// TIA Portal project "Anderca_Mihai_Teodor_Aplicatie_Practica_AIA_Licenta" (V15.1)

(* hardware
DEVICE "S7-1200 station_1"  S7-1200 Station
   slot 0: "Rack_0"  S7-1200 Rack  Rack  V1.0
   slot 1: "PLC_1"  CPU 1215C AC/DC/Rly  6ES7 215-1BG40-0XB0  V4.2
*)

// ===== PLC "PLC_1"  CPU 1215C AC/DC/Rly =====

VAR_GLOBAL   // PLC tag table "Palletizer tag table"
   "Transporto Role Incarcare Palet" AT %Q1.5 : Bool;
   "Tag_1" AT %M0.0 : Bool;
   "Senzor Palet Spate" AT %I5.2 : Bool;
   "Senzor Palet Fata" AT %I5.3 : Bool;
   "Lant Ascensor" AT %Q1.6 : Bool;
   "Senzor Palet Ridicat" AT %I5.6 : Bool;
   "Placa Deschisa" AT %M1.2 : Bool;
   "Palet Incarcat" AT %M1.4 : Bool;
   "Ascensor Ridicat" AT %Q1.7 : Bool;
   "Pusher" AT %Q2.1 : Bool;
   "Rand Complet Terminat" AT %M1.1 : Bool;
   "2 Cutii Incarcate" AT %M1.0 : Bool;
   "Banda Incarcare Cutii Incorporata" AT %Q2.3 : Bool;
   "Banda Incarcare Cutii" AT %Q2.5 : Bool;
   "Senzor Cutie Incarcata" AT %I5.4 : Bool;
   "Tag_6" AT %M0.3 : Bool;
   "Rand Incarcat" AT %M1.3 : Bool;
   "Tag_8" AT %M0.1 : Bool;
   "Cleste" AT %Q2.2 : Bool;
   "Deschidere Placa" AT %Q2.4 : Bool;
   "Placa Deschisa Maxim" AT %I5.5 : Bool;
   "Tag_9" AT %M0.4 : Bool;
   "Tag_10" AT %M1.6 : Bool;
   "Palet coborât" AT %M1.5 : Bool;
   "Coborare Palet" AT %Q2.0 : Bool;
   "Transportor Iesire" AT %Q2.6 : Bool;
   "Muta Ascensorul la Limita" AT %Q2.7 : Bool;
   "Tag_12" AT %M2.0 : Bool;
   "Tag_13" AT %M0.5 : Bool;
   "Tag_14" AT %M20.0 : Bool;
   "Placa Inchisa" AT %M3.0 : Bool;
   "Tag_16" AT %M3.1 : Bool;
   "Tag_17" AT %M3.2 : Bool;
   "Tag_18" AT %M0.6 : Bool;
   "Palet Gata de Coborâre" AT %M3.4 : Bool;
   "Palet Ridicat" AT %M3.6 : Bool;
END_VAR

VAR_GLOBAL   // PLC tag table "Sortare tag table"
   "Start Buton" AT %I4.0 : Bool;
   "Banda principala" AT %Q0.0 : Bool;
   "Banda Transportoare Stanga" AT %Q0.1 : Bool;
   "Banda Transportoare Dreapta" AT %Q0.2 : Bool;
   "Wheel Sorter" AT %Q0.4 : Bool;   // p
   "Deviere Stanga Wheel Sorter" AT %Q0.5 : Bool;
   "Deviere Dreapta Wheel Sorter" AT %Q0.6 : Bool;
   "Senzor cutie mica" AT %I4.1 : Bool;
   "Cutie Mica Detectata" AT %M30.0 : Bool;
   "Senzor Intrare Stanga" AT %I4.2 : Bool;
   "Cutie Mica Sortata" AT %M30.1 : Bool;
   "Senzor cutie mare" AT %I4.3 : Bool;
   "Senzor Intrare Dreapta" AT %I4.4 : Bool;
   "Cutie Mare Detectata" AT %M30.2 : Bool;
   "Cutie Mare Sortata" AT %M30.3 : Bool;
   "START" AT %M31.0 : Bool;
   "Start Led" AT %Q1.0 : Bool;
   "Stop Buton" AT %I4.5 : Bool;
   "STOP" AT %M31.1 : Bool;
   "Stop Led" AT %Q1.1 : Bool;
   "Banda Transportoare Inclinata" AT %Q0.7 : Bool;
END_VAR

VAR_GLOBAL CONSTANT   // PLC tag table "Sortare tag table"
   "None(1)" : Pip := 65535;
   "Automatic update(1)" : Pip := 0;
   "PIP 1(1)" : Pip := 1;
   "PIP 2(1)" : Pip := 2;
   "PIP 3(1)" : Pip := 3;
   "PIP 4(1)" : Pip := 4;
   "PIP OB Servo(1)" : Pip := 32768;
   "Local~MC(1)" : Hw_SubModule := 51;
   "Local~Common(1)" : Hw_SubModule := 50;
   "Local~Device(1)" : Hw_Device := 32;
   "Local~Configuration(1)" : Hw_SubModule := 33;
   "Local~Exec(1)" : Hw_SubModule := 52;
   "Local(1)" : Hw_SubModule := 49;
   "Local~PROFINET_interface_1(1)" : Hw_Interface := 64;
   "Local~PROFINET_interface_1~Port_1(1)" : Hw_Interface := 65;
   "Local~PROFINET_interface_1~Port_2(1)" : Hw_Interface := 66;
   "Local~HSC_1(1)" : Hw_Hsc := 257;
   "Local~HSC_2(1)" : Hw_Hsc := 258;
   "Local~HSC_3(1)" : Hw_Hsc := 259;
   "Local~HSC_4(1)" : Hw_Hsc := 260;
   "Local~HSC_5(1)" : Hw_Hsc := 261;
   "Local~HSC_6(1)" : Hw_Hsc := 262;
   "Local~AI_2_AQ_2_1(1)" : Hw_SubModule := 263;
   "Local~DI_14_DQ_10_1(1)" : Hw_SubModule := 264;
   "Local~Pulse_1(1)" : Hw_Pwm := 265;
   "Local~Pulse_2(1)" : Hw_Pwm := 266;
   "Local~Pulse_3(1)" : Hw_Pwm := 267;
   "Local~Pulse_4(1)" : Hw_Pwm := 268;
   "OB_Main(1)" : OB_PCYCLE := 1;
END_VAR

VAR_GLOBAL   // PLC tag table "PP tag table"
   "Senzor Amplasat" AT %I6.3 : Bool;
   "Senzor încorporat" AT %I6.4 : Bool;
   "Senzor Detecție Cutie deasupra Paletului" AT %I6.5 : Bool;
   "Transportor cu Role" AT %Q3.1 : Bool;
   "Prindere" AT %Q3.2 : Bool;
   "Deplasare Orizontală a Brațului" AT %Q3.3 : Bool;
   "Deplasare Verticală a Brațului" AT %Q3.4 : Bool;
   "Tag_7 pp" AT %M41.3 : Bool;
   "m41.4" AT %M41.5 : Bool;
   "Cutie detectată la Pick and Place" AT %M41.0 : Bool;
   "Tag_13 pp" AT %M41.1 : Bool;
   "Cutie Prinsă" AT %M41.2 : Bool;
   "Cutie deasupra Paletului" AT %M41.4 : Bool;
END_VAR

VAR_GLOBAL CONSTANT   // PLC tag table "PP tag table"
   "None(2)" : Pip := 65535;
   "Automatic update(2)" : Pip := 0;
   "PIP 1(2)" : Pip := 1;
   "PIP 2(2)" : Pip := 2;
   "PIP 3(2)" : Pip := 3;
   "PIP 4(2)" : Pip := 4;
   "PIP OB Servo(2)" : Pip := 32768;
   "Local~MC(2)" : Hw_SubModule := 51;
   "Local~Common(2)" : Hw_SubModule := 50;
   "Local~Device(2)" : Hw_Device := 32;
   "Local~Configuration(2)" : Hw_SubModule := 33;
   "Local~Exec(2)" : Hw_SubModule := 52;
   "Local(2)" : Hw_SubModule := 49;
   "Local~PROFINET_interface_1(2)" : Hw_Interface := 64;
   "Local~PROFINET_interface_1~Port_1(2)" : Hw_Interface := 65;
   "Local~PROFINET_interface_1~Port_2(2)" : Hw_Interface := 66;
   "Local~HSC_1(2)" : Hw_Hsc := 257;
   "Local~HSC_2(2)" : Hw_Hsc := 258;
   "Local~HSC_3(2)" : Hw_Hsc := 259;
   "Local~HSC_4(2)" : Hw_Hsc := 260;
   "Local~HSC_5(2)" : Hw_Hsc := 261;
   "Local~HSC_6(2)" : Hw_Hsc := 262;
   "Local~AI_2_AQ_2_1(2)" : Hw_SubModule := 263;
   "Local~DI_14_DQ_10_1(2)" : Hw_SubModule := 264;
   "Local~Pulse_1(2)" : Hw_Pwm := 265;
   "Local~Pulse_2(2)" : Hw_Pwm := 266;
   "Local~Pulse_3(2)" : Hw_Pwm := 267;
   "Local~Pulse_4(2)" : Hw_Pwm := 268;
   "OB_Main(2)" : OB_PCYCLE := 1;
END_VAR

// folder: System blocks/Program resources

DATA_BLOCK "IEC_Timer_0_DB"   // DB1
{ S7_Optimized_Access := 'TRUE' }
AUTHOR : Simatic
FAMILY : IEC
NAME : IEC_TMR
VERSION : 1.0
// stored: InstanceOfName IEC_TIMER
"IEC_TIMER"
BEGIN
END_DATA_BLOCK

DATA_BLOCK "IEC_Timer_0_DB_2"   // DB2
{ S7_Optimized_Access := 'TRUE' }
AUTHOR : Simatic
FAMILY : IEC
NAME : IEC_TMR
VERSION : 1.0
// stored: InstanceOfName IEC_TIMER
"IEC_TIMER"
BEGIN
END_DATA_BLOCK

DATA_BLOCK "IEC_Counter_0_DB"   // DB3
{ S7_Optimized_Access := 'TRUE' }
AUTHOR : Simatic
FAMILY : IEC
NAME : CNTR
VERSION : 1.0
// stored: InstanceOfName IEC_COUNTER
"IEC_COUNTER"
BEGIN
END_DATA_BLOCK

DATA_BLOCK "IEC_Timer_0_DB_1"   // DB4
{ S7_Optimized_Access := 'TRUE' }
AUTHOR : Simatic
FAMILY : IEC
NAME : IEC_TMR
VERSION : 1.0
// stored: InstanceOfName IEC_TIMER
"IEC_TIMER"
BEGIN
END_DATA_BLOCK

DATA_BLOCK "IEC_Counter_0_DB_1"   // DB5
{ S7_Optimized_Access := 'TRUE' }
AUTHOR : Simatic
FAMILY : IEC
NAME : CNTR
VERSION : 1.0
// stored: InstanceOfName IEC_COUNTER
"IEC_COUNTER"
BEGIN
END_DATA_BLOCK

DATA_BLOCK "IEC_Timer_0_DB_3"   // DB6
{ S7_Optimized_Access := 'TRUE' }
AUTHOR : Simatic
FAMILY : IEC
NAME : IEC_TMR
VERSION : 1.0
// stored: InstanceOfName IEC_TIMER
"IEC_TIMER"
BEGIN
END_DATA_BLOCK

DATA_BLOCK "IEC_Timer_0_DB_4"   // DB7
{ S7_Optimized_Access := 'TRUE' }
AUTHOR : Simatic
FAMILY : IEC
NAME : IEC_TMR
VERSION : 1.0
// stored: InstanceOfName IEC_TIMER
"IEC_TIMER"
BEGIN
END_DATA_BLOCK

DATA_BLOCK "IEC_Timer_0_DB_5"   // DB8
{ S7_Optimized_Access := 'TRUE' }
AUTHOR : Simatic
FAMILY : IEC
NAME : IEC_TMR
VERSION : 1.0
// stored: InstanceOfName IEC_TIMER
"IEC_TIMER"
BEGIN
END_DATA_BLOCK

DATA_BLOCK "IEC_Timer_0_DB_6"   // DB9
{ S7_Optimized_Access := 'TRUE' }
AUTHOR : Simatic
FAMILY : IEC
NAME : IEC_TMR
VERSION : 1.0
// stored: InstanceOfName IEC_TIMER
"IEC_TIMER"
BEGIN
END_DATA_BLOCK

DATA_BLOCK "IEC_Counter_0_DB_2"   // DB10
{ S7_Optimized_Access := 'TRUE' }
AUTHOR : Simatic
FAMILY : IEC
NAME : CNTR
VERSION : 1.0
// stored: InstanceOfName IEC_COUNTER
"IEC_COUNTER"
BEGIN
END_DATA_BLOCK

DATA_BLOCK "IEC_Timer_0_DB_7"   // DB11
{ S7_Optimized_Access := 'TRUE' }
AUTHOR : Simatic
FAMILY : IEC
NAME : IEC_TMR
VERSION : 1.0
// stored: InstanceOfName IEC_TIMER
"IEC_TIMER"
BEGIN
END_DATA_BLOCK

DATA_BLOCK "IEC_Timer_0_DB_8"   // DB12
{ S7_Optimized_Access := 'TRUE' }
AUTHOR : Simatic
FAMILY : IEC
NAME : IEC_TMR
VERSION : 1.0
// stored: InstanceOfName IEC_TIMER
"IEC_TIMER"
BEGIN
END_DATA_BLOCK

DATA_BLOCK "IEC_Timer_0_DB_9"   // DB13
{ S7_Optimized_Access := 'TRUE' }
AUTHOR : Simatic
FAMILY : IEC
NAME : IEC_TMR
VERSION : 1.0
// stored: InstanceOfName IEC_TIMER
"IEC_TIMER"
BEGIN
END_DATA_BLOCK

DATA_BLOCK "IEC_Timer_0_DB_10"   // DB14
{ S7_Optimized_Access := 'TRUE' }
AUTHOR : Simatic
FAMILY : IEC
NAME : IEC_TMR
VERSION : 1.0
// stored: InstanceOfName IEC_TIMER
"IEC_TIMER"
BEGIN
END_DATA_BLOCK

DATA_BLOCK "IEC_Timer_0_DB_11"   // DB15
{ S7_Optimized_Access := 'TRUE' }
AUTHOR : Simatic
FAMILY : IEC
NAME : IEC_TMR
VERSION : 1.0
// stored: InstanceOfName IEC_TIMER
"IEC_TIMER"
BEGIN
END_DATA_BLOCK

DATA_BLOCK "IEC_Timer_0_DB_12"   // DB16
{ S7_Optimized_Access := 'TRUE' }
AUTHOR : Simatic
FAMILY : IEC
NAME : IEC_TMR
VERSION : 1.0
// stored: InstanceOfName IEC_TIMER
"IEC_TIMER"
BEGIN
END_DATA_BLOCK

// folder: (top level)

FUNCTION "MHJ-PLC-Lab-Function-S71200" : Void   // FC9000, SCL
{ S7_Optimized_Access := 'TRUE' }
VERSION : 0.1
   VAR_TEMP
      rdTimeReturn : Int;
      outputTime : DTL;
      SyncVal : Byte;
      forVal : Int;
      forVal_2 : Int;
      Value : Byte;
   END_VAR
   VAR CONSTANT
      CompVal : Byte := 16#34;
      Value_01 : Byte := 16#11;
      Value_01_DW : DWord := 16#A165_D992;
      Value_02_DW : DWord := 16#58BE_4401;
   END_VAR
BEGIN

   #Value:=PEEK(area := 16#82,
        dbNumber := 0,
        byteOffset := 511);
   #Value := #Value + 1;

   POKE(area := 16#82,
        dbNumber := 0,
        byteOffset := 511,
        value := #Value);

   POKE(area:=16#81,
        dbNumber:=0,
        byteOffset:=1016,
        value:=#Value_01_DW);
   POKE(area := 16#81,
        dbNumber := 0,
        byteOffset := 1020,
        value := #Value_02_DW);

   POKE(area := 16#81,
        dbNumber := 0,
        byteOffset := 511,
        value := B#16#00);

   FOR #forVal := 0 TO 120 DO
       FOR #forVal_2:=0 TO 10 DO
           #rdTimeReturn:=RD_SYS_T(#outputTime);
           #rdTimeReturn := WR_SYS_T(#outputTime);
           #rdTimeReturn := RD_SYS_T(#outputTime);
           #rdTimeReturn := WR_SYS_T(#outputTime);
       END_FOR;
       #SyncVal:= PEEK(area := 16#81,
                      dbNumber := 0,
                      byteOffset := 511);
       IF #SyncVal = #CompVal THEN
          GOTO M_1;
       END_IF;
   END_FOR;
   RETURN;

   M_1:
   POKE(area := 16#81,
        dbNumber := 0,
        byteOffset := 511,
        value := B#16#0);
END_FUNCTION

ORGANIZATION_BLOCK "Main"   // OB1, LAD, ProgramCycle
TITLE = "Main Program Sweep (Cycle)"
{ S7_Optimized_Access := 'TRUE' }
VERSION : 0.1
   VAR_INPUT
      Initial_Call : Bool;   // Initial call of this OB
      Remanence : Bool;   // =True, if remanent data are available
   END_VAR
   VAR_TEMP
      Time1 : Time;
   END_VAR
   VAR_TEMP   // added for the SCL form of the ladder/FBD networks
      _w1 : Bool;
      _w2 : Bool;
   END_VAR
BEGIN

REGION Network 1
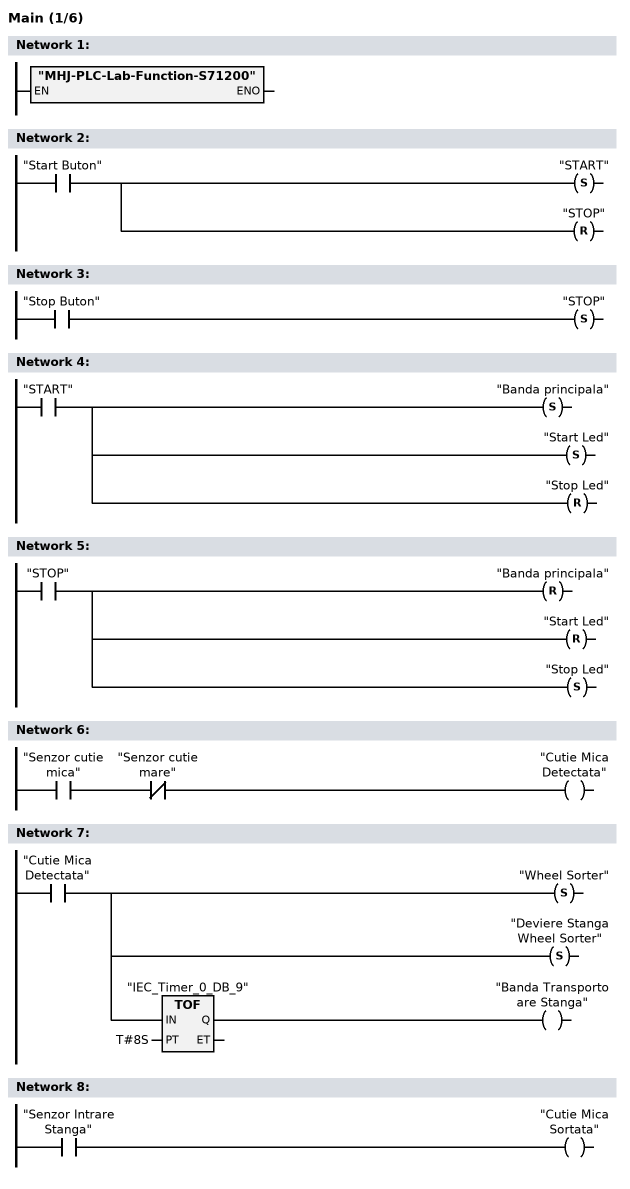
   RUNG wire#powerrail
      "MHJ-PLC-Lab-Function-S71200"()
   END_RUNG
   // the same network as SCL:
   "MHJ-PLC-Lab-Function-S71200"();
END_REGION

REGION Network 2
   RUNG wire#powerrail
      Contact( "Start Buton" )
      wire#w1
      S_Coil( "START" )
   END_RUNG
   RUNG wire#w1
      R_Coil( "STOP" )
   END_RUNG
   // the same network as SCL:
   IF "Start Buton" THEN
       "START" := TRUE;
       "STOP" := FALSE;
   END_IF;
END_REGION

REGION Network 3
   RUNG wire#powerrail
      Contact( "Stop Buton" )
      S_Coil( "STOP" )
   END_RUNG
   // the same network as SCL:
   IF "Stop Buton" THEN "STOP" := TRUE; END_IF;
END_REGION

REGION Network 4
   RUNG wire#powerrail
      Contact( "START" )
      wire#w1
      S_Coil( "Banda principala" )
   END_RUNG
   RUNG wire#w1
      S_Coil( "Start Led" )
   END_RUNG
   RUNG wire#w1
      R_Coil( "Stop Led" )
   END_RUNG
   // the same network as SCL:
   IF "START" THEN
       "Banda principala" := TRUE;
       "Start Led" := TRUE;
       "Stop Led" := FALSE;
   END_IF;
END_REGION

REGION Network 5
   RUNG wire#powerrail
      Contact( "STOP" )
      wire#w1
      R_Coil( "Banda principala" )
   END_RUNG
   RUNG wire#w1
      R_Coil( "Start Led" )
   END_RUNG
   RUNG wire#w1
      S_Coil( "Stop Led" )
   END_RUNG
   // the same network as SCL:
   IF "STOP" THEN
       "Banda principala" := FALSE;
       "Start Led" := FALSE;
       "Stop Led" := TRUE;
   END_IF;
END_REGION

REGION Network 6
   RUNG wire#powerrail
      Contact( "Senzor cutie mica" )
      I_Contact( "Senzor cutie mare" )
      Coil( "Cutie Mica Detectata" )
   END_RUNG
   // the same network as SCL:
   "Cutie Mica Detectata" := "Senzor cutie mica" AND NOT "Senzor cutie mare";
END_REGION

REGION Network 7
   IF "Cutie Mica Detectata" THEN
       "Wheel Sorter" := TRUE;
       "Deviere Stanga Wheel Sorter" := TRUE;
   END_IF;
   "IEC_Timer_0_DB_9".TOF(IN := "Cutie Mica Detectata", PT := T#8S);
   "Banda Transportoare Stanga" := "IEC_Timer_0_DB_9".Q;
END_REGION

REGION Network 8
   RUNG wire#powerrail
      Contact( "Senzor Intrare Stanga" )
      Coil( "Cutie Mica Sortata" )
   END_RUNG
   // the same network as SCL:
   "Cutie Mica Sortata" := "Senzor Intrare Stanga";
END_REGION

REGION Network 9: p
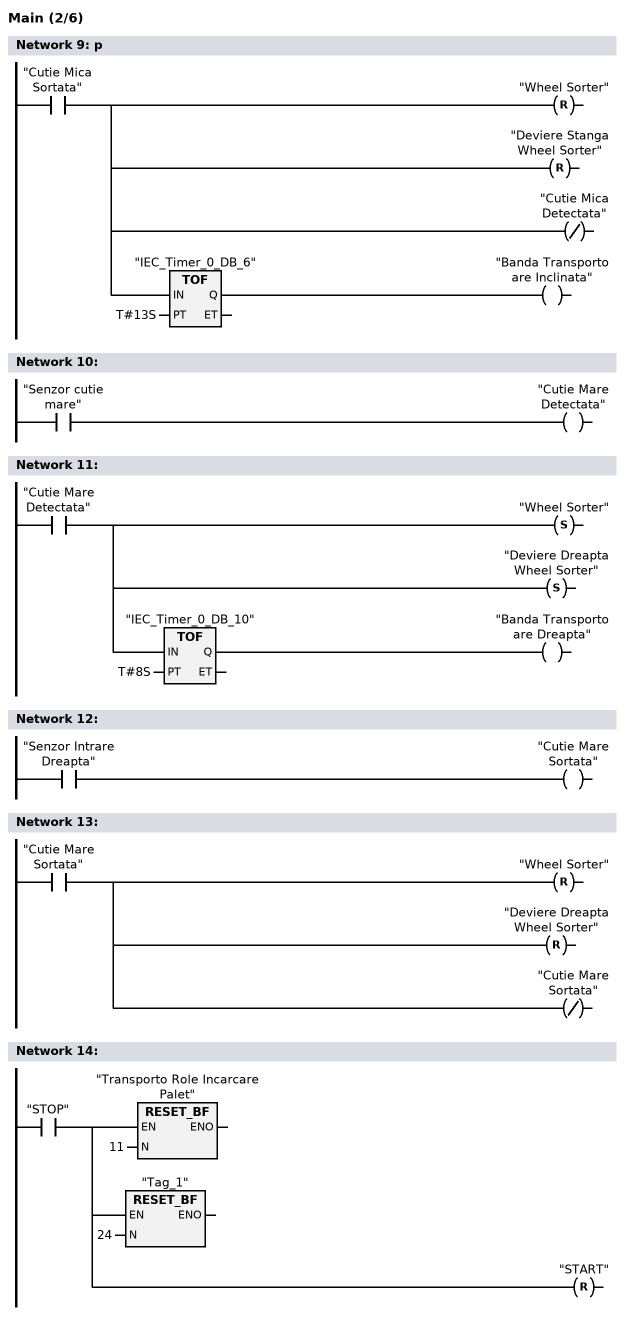
   IF "Cutie Mica Sortata" THEN
       "Wheel Sorter" := FALSE;
       "Deviere Stanga Wheel Sorter" := FALSE;
   END_IF;
   "Cutie Mica Detectata" := NOT "Cutie Mica Sortata";
   "IEC_Timer_0_DB_6".TOF(IN := "Cutie Mica Sortata", PT := T#13S);
   "Banda Transportoare Inclinata" := "IEC_Timer_0_DB_6".Q;
END_REGION

REGION Network 10
   RUNG wire#powerrail
      Contact( "Senzor cutie mare" )
      Coil( "Cutie Mare Detectata" )
   END_RUNG
   // the same network as SCL:
   "Cutie Mare Detectata" := "Senzor cutie mare";
END_REGION

REGION Network 11
   IF "Cutie Mare Detectata" THEN
       "Wheel Sorter" := TRUE;
       "Deviere Dreapta Wheel Sorter" := TRUE;
   END_IF;
   "IEC_Timer_0_DB_10".TOF(IN := "Cutie Mare Detectata", PT := T#8S);
   "Banda Transportoare Dreapta" := "IEC_Timer_0_DB_10".Q;
END_REGION

REGION Network 12
   RUNG wire#powerrail
      Contact( "Senzor Intrare Dreapta" )
      Coil( "Cutie Mare Sortata" )
   END_RUNG
   // the same network as SCL:
   "Cutie Mare Sortata" := "Senzor Intrare Dreapta";
END_REGION

REGION Network 13
   RUNG wire#powerrail
      Contact( "Cutie Mare Sortata" )
      wire#w1
      R_Coil( "Wheel Sorter" )
   END_RUNG
   RUNG wire#w1
      R_Coil( "Deviere Dreapta Wheel Sorter" )
   END_RUNG
   RUNG wire#w1
      I_Coil( "Cutie Mare Sortata" )
   END_RUNG
   // the same network as SCL:
   IF "Cutie Mare Sortata" THEN
       "Wheel Sorter" := FALSE;
       "Deviere Dreapta Wheel Sorter" := FALSE;
   END_IF;
   "Cutie Mare Sortata" := NOT "Cutie Mare Sortata";
END_REGION

REGION Network 14
   // no SCL statement known for RBitfield: written as a call
   #_w1 := "STOP";
   IF #_w1 THEN
       RESET_BF(operand := "Transporto Role Incarcare Palet", n := 11);
       RESET_BF(operand := "Tag_1", n := 24);
       "START" := FALSE;
   END_IF;
END_REGION

REGION Network 15
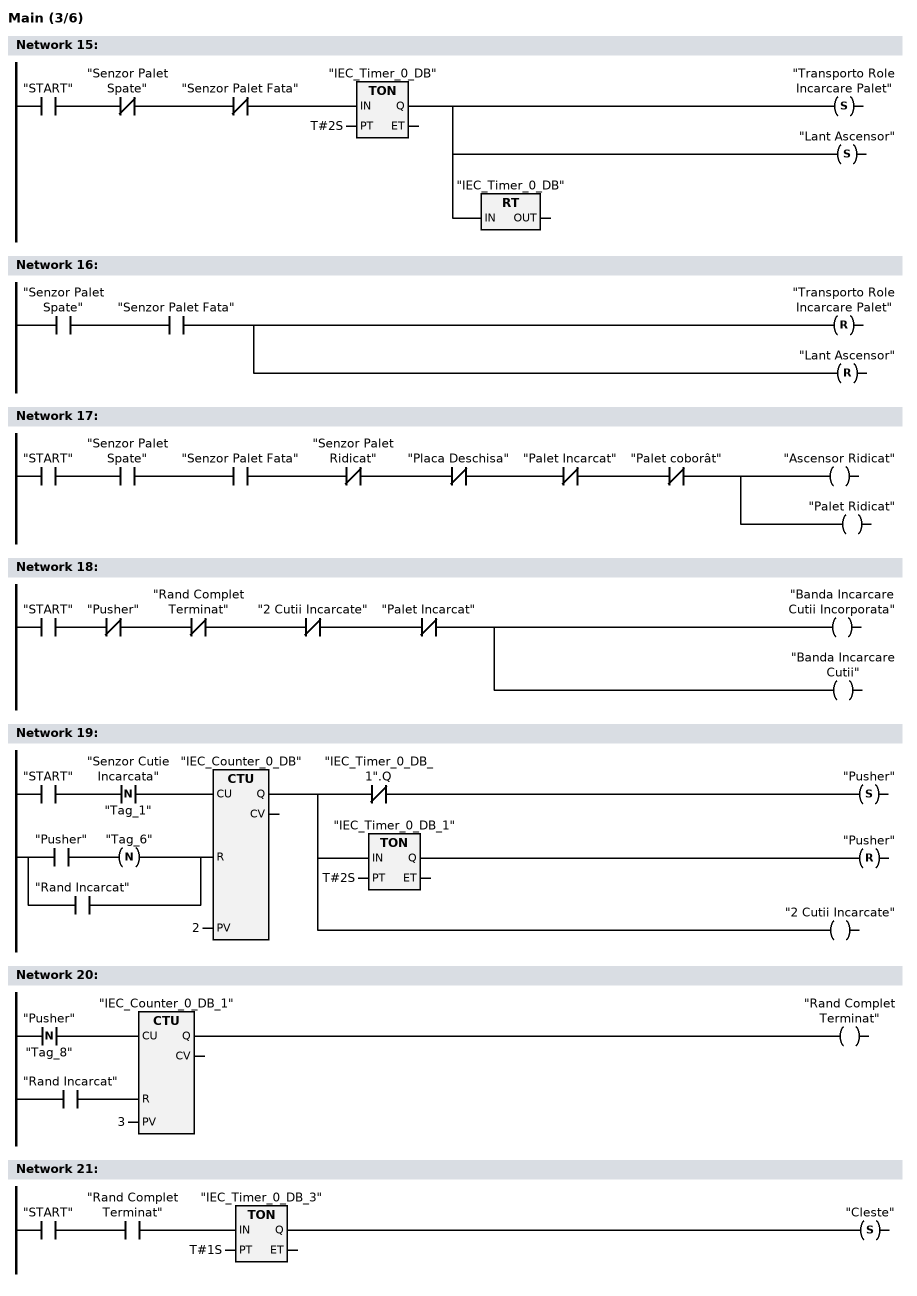
   "IEC_Timer_0_DB".TON(IN := "START" AND NOT "Senzor Palet Spate" AND NOT "Senzor Palet Fata", PT := T#2S);
   IF "IEC_Timer_0_DB".Q THEN
       "Transporto Role Incarcare Palet" := TRUE;
       "Lant Ascensor" := TRUE;
       RESET_TIMER("IEC_Timer_0_DB");
   END_IF;
END_REGION

REGION Network 16
   RUNG wire#powerrail
      Contact( "Senzor Palet Spate" )
      Contact( "Senzor Palet Fata" )
      wire#w1
      R_Coil( "Transporto Role Incarcare Palet" )
   END_RUNG
   RUNG wire#w1
      R_Coil( "Lant Ascensor" )
   END_RUNG
   // the same network as SCL:
   IF "Senzor Palet Spate" AND "Senzor Palet Fata" THEN
       "Transporto Role Incarcare Palet" := FALSE;
       "Lant Ascensor" := FALSE;
   END_IF;
END_REGION

REGION Network 17
   RUNG wire#powerrail
      Contact( "START" )
      Contact( "Senzor Palet Spate" )
      Contact( "Senzor Palet Fata" )
      I_Contact( "Senzor Palet Ridicat" )
      I_Contact( "Placa Deschisa" )
      I_Contact( "Palet Incarcat" )
      I_Contact( "Palet coborât" )
      wire#w1
      Coil( "Ascensor Ridicat" )
   END_RUNG
   RUNG wire#w1
      Coil( "Palet Ridicat" )
   END_RUNG
   // the same network as SCL:
   "Ascensor Ridicat" := "START" AND "Senzor Palet Spate" AND "Senzor Palet Fata" AND NOT "Senzor Palet Ridicat" AND NOT "Placa Deschisa" AND NOT "Palet Incarcat" AND NOT "Palet coborât";
   "Palet Ridicat" := "Ascensor Ridicat";
END_REGION

REGION Network 18
   RUNG wire#powerrail
      Contact( "START" )
      I_Contact( "Pusher" )
      I_Contact( "Rand Complet Terminat" )
      I_Contact( "2 Cutii Incarcate" )
      I_Contact( "Palet Incarcat" )
      wire#w1
      Coil( "Banda Incarcare Cutii Incorporata" )
   END_RUNG
   RUNG wire#w1
      Coil( "Banda Incarcare Cutii" )
   END_RUNG
   // the same network as SCL:
   "Banda Incarcare Cutii Incorporata" := "START" AND NOT "Pusher" AND NOT "Rand Complet Terminat" AND NOT "2 Cutii Incarcate" AND NOT "Palet Incarcat";
   "Banda Incarcare Cutii" := "Banda Incarcare Cutii Incorporata";
END_REGION

REGION Network 19
   #_w1 := "START" AND NOT "Senzor Cutie Incarcata" AND "Tag_1";   // falling edge of "Senzor Cutie Incarcata"
   "Tag_1" := "Senzor Cutie Incarcata";
   #_w2 := NOT "Pusher" AND "Tag_6";   // falling edge
   "Tag_6" := "Pusher";
   "IEC_Counter_0_DB".CTU(CU := #_w1, R := #_w2 OR "Rand Incarcat", PV := 2);
   IF "IEC_Counter_0_DB".Q AND NOT "IEC_Timer_0_DB_1".Q THEN "Pusher" := TRUE; END_IF;
   "IEC_Timer_0_DB_1".TON(IN := "IEC_Counter_0_DB".Q, PT := T#2S);
   IF "IEC_Timer_0_DB_1".Q THEN "Pusher" := FALSE; END_IF;
   "2 Cutii Incarcate" := "IEC_Counter_0_DB".Q;
END_REGION

REGION Network 20
   #_w1 := NOT "Pusher" AND "Tag_8";   // falling edge of "Pusher"
   "Tag_8" := "Pusher";
   "IEC_Counter_0_DB_1".CTU(CU := #_w1, R := "Rand Incarcat", PV := 3);
   "Rand Complet Terminat" := "IEC_Counter_0_DB_1".Q;
END_REGION

REGION Network 21
   "IEC_Timer_0_DB_3".TON(IN := "START" AND "Rand Complet Terminat", PT := T#1S);
   IF "IEC_Timer_0_DB_3".Q THEN "Cleste" := TRUE; END_IF;
END_REGION

REGION Network 22
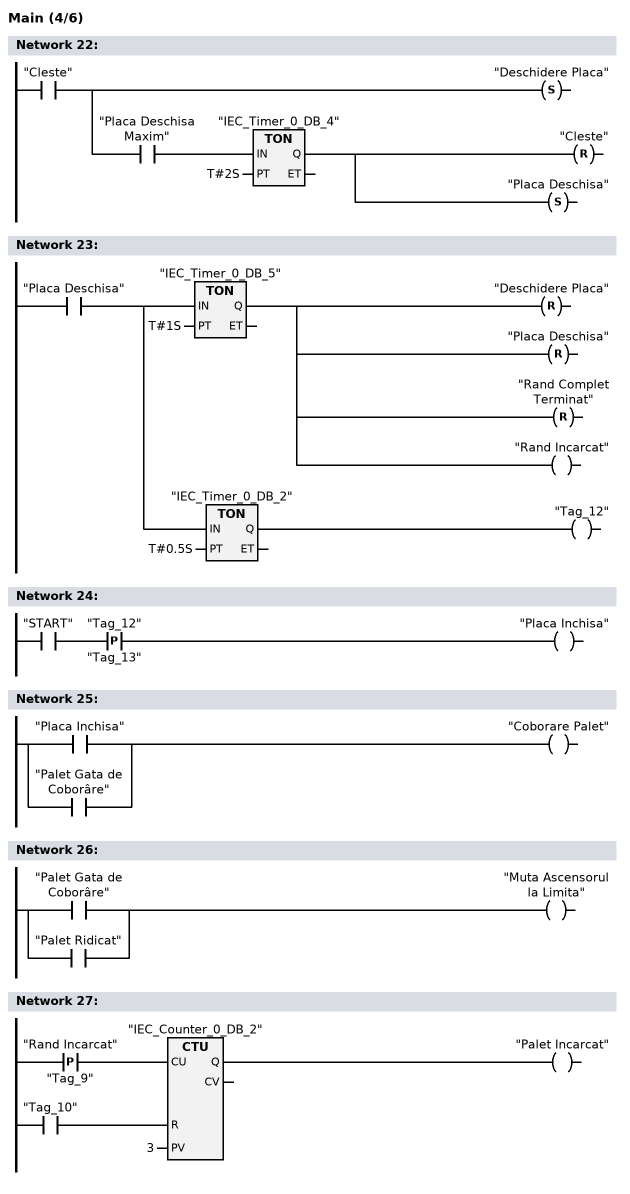
   IF "Cleste" THEN "Deschidere Placa" := TRUE; END_IF;
   "IEC_Timer_0_DB_4".TON(IN := "Cleste" AND "Placa Deschisa Maxim", PT := T#2S);
   IF "IEC_Timer_0_DB_4".Q THEN
       "Cleste" := FALSE;
       "Placa Deschisa" := TRUE;
   END_IF;
END_REGION

REGION Network 23
   "IEC_Timer_0_DB_5".TON(IN := "Placa Deschisa", PT := T#1S);
   IF "IEC_Timer_0_DB_5".Q THEN "Deschidere Placa" := FALSE; END_IF;
   #_w1 := "Placa Deschisa";
   IF "IEC_Timer_0_DB_5".Q THEN
       "Placa Deschisa" := FALSE;
       "Rand Complet Terminat" := FALSE;
   END_IF;
   "Rand Incarcat" := "IEC_Timer_0_DB_5".Q;
   "IEC_Timer_0_DB_2".TON(IN := #_w1, PT := T#0.5S);
   "Tag_12" := "IEC_Timer_0_DB_2".Q;
END_REGION

REGION Network 24
   RUNG wire#powerrail
      Contact( "START" )
      P_Contact(operand := "Tag_12", bit := "Tag_13")
      Coil( "Placa Inchisa" )
   END_RUNG
   // the same network as SCL:
   #_w1 := "START" AND "Tag_12" AND NOT "Tag_13";   // rising edge of "Tag_12"
   "Tag_13" := "Tag_12";
   "Placa Inchisa" := #_w1;
END_REGION

REGION Network 25
   RUNG wire#powerrail
      Contact( "Placa Inchisa" )
      wire#w1
      Coil( "Coborare Palet" )
   END_RUNG
   RUNG wire#powerrail
      Contact( "Palet Gata de Coborâre" )
   END_RUNG wire#w1
   // the same network as SCL:
   "Coborare Palet" := "Placa Inchisa" OR "Palet Gata de Coborâre";
END_REGION

REGION Network 26
   RUNG wire#powerrail
      Contact( "Palet Gata de Coborâre" )
      wire#w1
      Coil( "Muta Ascensorul la Limita" )
   END_RUNG
   RUNG wire#powerrail
      Contact( "Palet Ridicat" )
   END_RUNG wire#w1
   // the same network as SCL:
   "Muta Ascensorul la Limita" := "Palet Gata de Coborâre" OR "Palet Ridicat";
END_REGION

REGION Network 27
   #_w1 := "Rand Incarcat" AND NOT "Tag_9";   // rising edge of "Rand Incarcat"
   "Tag_9" := "Rand Incarcat";
   "IEC_Counter_0_DB_2".CTU(CU := #_w1, R := "Tag_10", PV := 3);
   "Palet Incarcat" := "IEC_Counter_0_DB_2".Q;
END_REGION

REGION Network 28
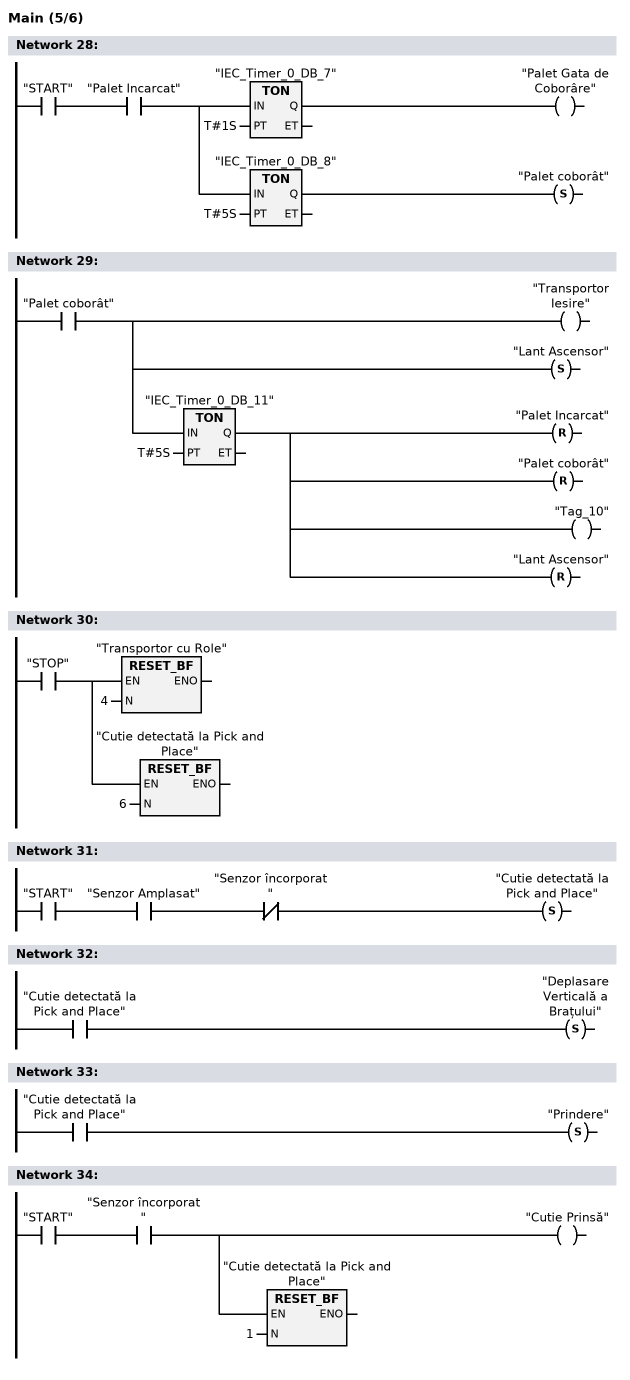
   #_w1 := "START" AND "Palet Incarcat";
   "IEC_Timer_0_DB_7".TON(IN := #_w1, PT := T#1S);
   "Palet Gata de Coborâre" := "IEC_Timer_0_DB_7".Q;
   "IEC_Timer_0_DB_8".TON(IN := #_w1, PT := T#5S);
   IF "IEC_Timer_0_DB_8".Q THEN "Palet coborât" := TRUE; END_IF;
END_REGION

REGION Network 29
   "Transportor Iesire" := "Palet coborât";
   IF "Palet coborât" THEN "Lant Ascensor" := TRUE; END_IF;
   "IEC_Timer_0_DB_11".TON(IN := "Palet coborât", PT := T#5S);
   IF "IEC_Timer_0_DB_11".Q THEN
       "Palet Incarcat" := FALSE;
       "Palet coborât" := FALSE;
   END_IF;
   "Tag_10" := "IEC_Timer_0_DB_11".Q;
   IF "IEC_Timer_0_DB_11".Q THEN "Lant Ascensor" := FALSE; END_IF;
END_REGION

REGION Network 30
   // no SCL statement known for RBitfield: written as a call
   #_w1 := "STOP";
   IF #_w1 THEN
       RESET_BF(operand := "Transportor cu Role", n := 4);
       RESET_BF(operand := "Cutie detectată la Pick and Place", n := 6);
   END_IF;
END_REGION

REGION Network 31
   RUNG wire#powerrail
      Contact( "START" )
      Contact( "Senzor Amplasat" )
      I_Contact( "Senzor încorporat" )
      S_Coil( "Cutie detectată la Pick and Place" )
   END_RUNG
   // the same network as SCL:
   IF "START" AND "Senzor Amplasat" AND NOT "Senzor încorporat" THEN
       "Cutie detectată la Pick and Place" := TRUE;
   END_IF;
END_REGION

REGION Network 32
   RUNG wire#powerrail
      Contact( "Cutie detectată la Pick and Place" )
      S_Coil( "Deplasare Verticală a Brațului" )
   END_RUNG
   // the same network as SCL:
   IF "Cutie detectată la Pick and Place" THEN "Deplasare Verticală a Brațului" := TRUE; END_IF;
END_REGION

REGION Network 33
   RUNG wire#powerrail
      Contact( "Cutie detectată la Pick and Place" )
      S_Coil( "Prindere" )
   END_RUNG
   // the same network as SCL:
   IF "Cutie detectată la Pick and Place" THEN "Prindere" := TRUE; END_IF;
END_REGION

REGION Network 34
   // no SCL statement known for RBitfield: written as a call
   "Cutie Prinsă" := "START" AND "Senzor încorporat";
   IF "Cutie Prinsă" THEN RESET_BF(operand := "Cutie detectată la Pick and Place", n := 1); END_IF;
END_REGION

REGION Network 35
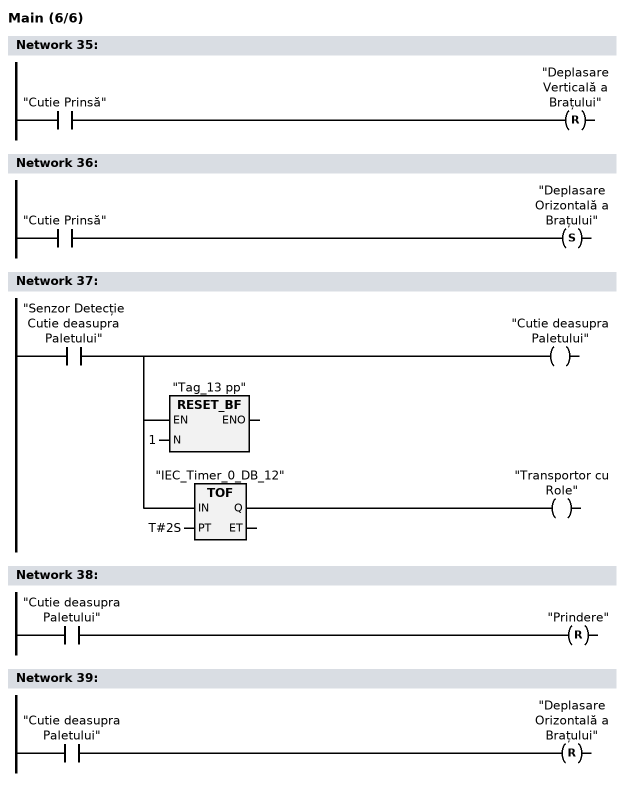
   RUNG wire#powerrail
      Contact( "Cutie Prinsă" )
      R_Coil( "Deplasare Verticală a Brațului" )
   END_RUNG
   // the same network as SCL:
   IF "Cutie Prinsă" THEN "Deplasare Verticală a Brațului" := FALSE; END_IF;
END_REGION

REGION Network 36
   RUNG wire#powerrail
      Contact( "Cutie Prinsă" )
      S_Coil( "Deplasare Orizontală a Brațului" )
   END_RUNG
   // the same network as SCL:
   IF "Cutie Prinsă" THEN "Deplasare Orizontală a Brațului" := TRUE; END_IF;
END_REGION

REGION Network 37
   // no SCL statement known for RBitfield: written as a call
   "Cutie deasupra Paletului" := "Senzor Detecție Cutie deasupra Paletului";
   #_w1 := "Senzor Detecție Cutie deasupra Paletului";
   IF #_w1 THEN RESET_BF(operand := "Tag_13 pp", n := 1); END_IF;
   "IEC_Timer_0_DB_12".TOF(IN := #_w1, PT := T#2S);
   "Transportor cu Role" := "IEC_Timer_0_DB_12".Q;
END_REGION

REGION Network 38
   RUNG wire#powerrail
      Contact( "Cutie deasupra Paletului" )
      R_Coil( "Prindere" )
   END_RUNG
   // the same network as SCL:
   IF "Cutie deasupra Paletului" THEN "Prindere" := FALSE; END_IF;
END_REGION

REGION Network 39
   RUNG wire#powerrail
      Contact( "Cutie deasupra Paletului" )
      R_Coil( "Deplasare Orizontală a Brațului" )
   END_RUNG
   // the same network as SCL:
   IF "Cutie deasupra Paletului" THEN "Deplasare Orizontală a Brațului" := FALSE; END_IF;
END_REGION
END_ORGANIZATION_BLOCK